// Mitsubishi GX Works2 project: GPF-73G-N2-21110030(220208)   PLC: Q02U

PROGRAM OVEN
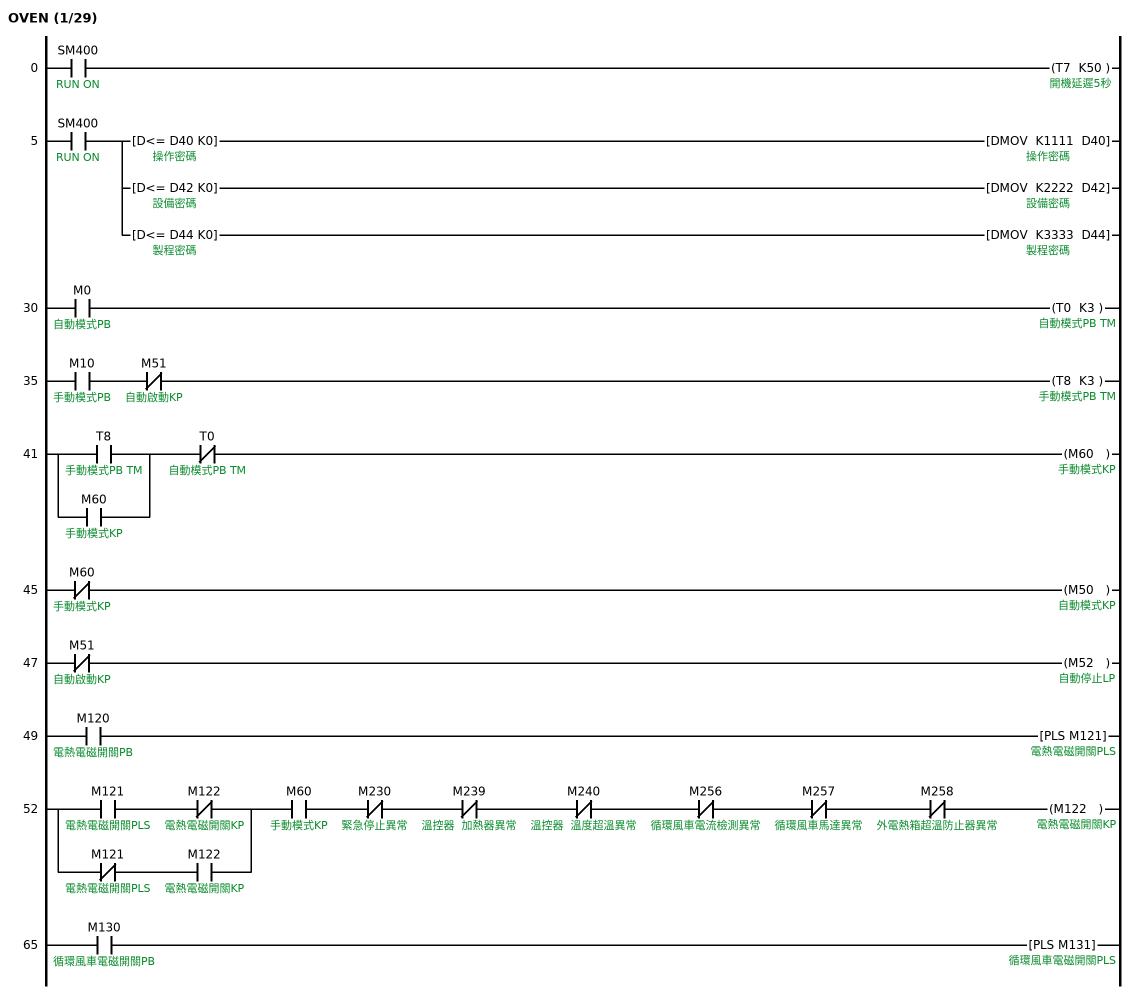
0     LD      SM400  ; RUN ON
      OUT     T7 K50  ; 開機延遲5秒
5     LD      SM400  ; RUN ON
      MPS
      ANDD<=  D40 K0  ; 操作密碼
      DMOV    K1111 D40
      MRD
      ANDD<=  D42 K0  ; 設備密碼
      DMOV    K2222 D42
      MPP
      ANDD<=  D44 K0  ; 製程密碼
      DMOV    K3333 D44
30    LD      M0  ; 自動模式PB
      OUT     T0 K3  ; 自動模式PB TM
35    LD      M10  ; 手動模式PB
      ANI     M51  ; 自動啟動KP
      OUT     T8 K3  ; 手動模式PB TM
41    LD      T8  ; 手動模式PB TM
      OR      M60  ; 手動模式KP
      ANI     T0  ; 自動模式PB TM
      OUT     M60  ; 手動模式KP
45    LDI     M60  ; 手動模式KP
      OUT     M50  ; 自動模式KP
47    LDI     M51  ; 自動啟動KP
      OUT     M52  ; 自動停止LP
49    LD      M120  ; 電熱電磁開關PB
      PLS     M121  ; 電熱電磁開關PLS
52    LD      M121  ; 電熱電磁開關PLS
      ANI     M122  ; 電熱電磁開關KP
      LDI     M121  ; 電熱電磁開關PLS
      AND     M122  ; 電熱電磁開關KP
      ORB
      AND     M60  ; 手動模式KP
      ANI     M230  ; 緊急停止異常
      ANI     M239  ; 溫控器  加熱器異常
      ANI     M240  ; 溫控器  溫度超溫異常
      ANI     M256  ; 循環風車電流檢測異常
      ANI     M257  ; 循環風車馬達異常
      ANI     M258  ; 外電熱箱超溫防止器異常
      OUT     M122  ; 電熱電磁開關KP
65    LD      M130  ; 循環風車電磁開關PB
      PLS     M131  ; 循環風車電磁開關PLS
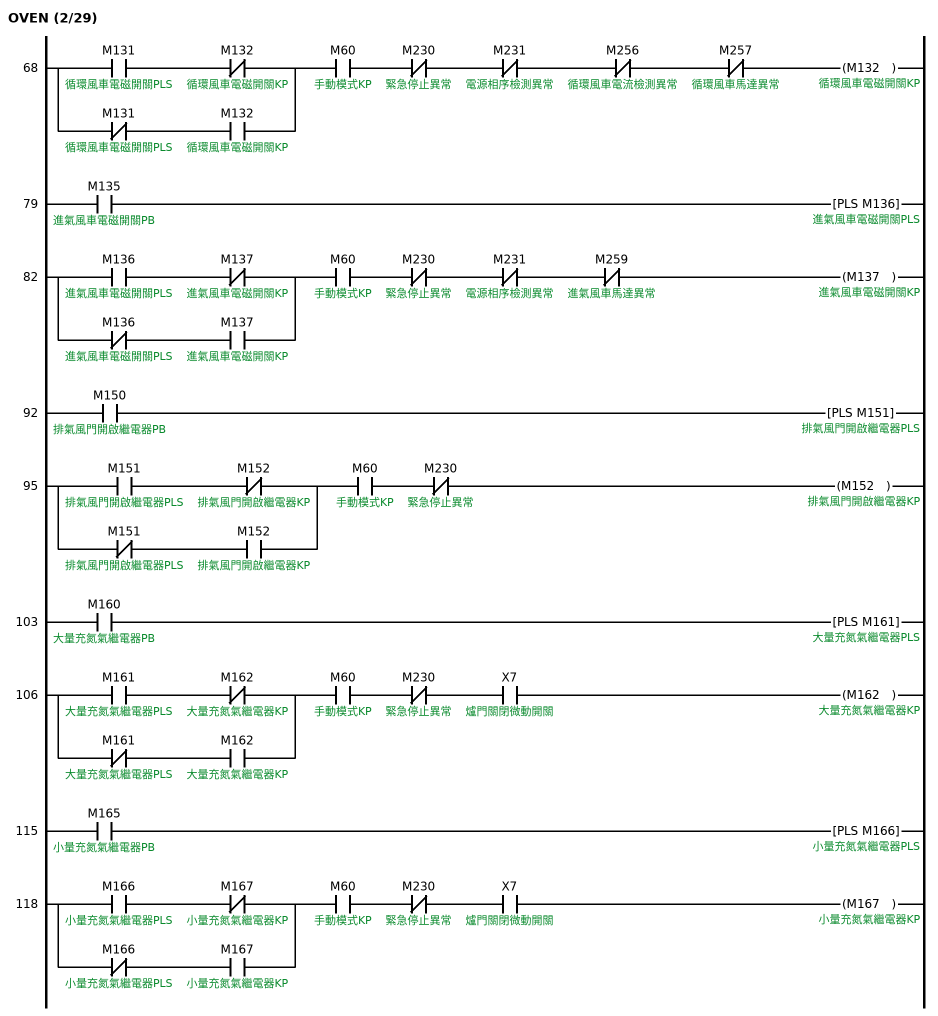
68    LD      M131  ; 循環風車電磁開關PLS
      ANI     M132  ; 循環風車電磁開關KP
      LDI     M131  ; 循環風車電磁開關PLS
      AND     M132  ; 循環風車電磁開關KP
      ORB
      AND     M60  ; 手動模式KP
      ANI     M230  ; 緊急停止異常
      ANI     M231  ; 電源相序檢測異常
      ANI     M256  ; 循環風車電流檢測異常
      ANI     M257  ; 循環風車馬達異常
      OUT     M132  ; 循環風車電磁開關KP
79    LD      M135  ; 進氣風車電磁開關PB
      PLS     M136  ; 進氣風車電磁開關PLS
82    LD      M136  ; 進氣風車電磁開關PLS
      ANI     M137  ; 進氣風車電磁開關KP
      LDI     M136  ; 進氣風車電磁開關PLS
      AND     M137  ; 進氣風車電磁開關KP
      ORB
      AND     M60  ; 手動模式KP
      ANI     M230  ; 緊急停止異常
      ANI     M231  ; 電源相序檢測異常
      ANI     M259  ; 進氣風車馬達異常
      OUT     M137  ; 進氣風車電磁開關KP
92    LD      M150  ; 排氣風門開啟繼電器PB
      PLS     M151  ; 排氣風門開啟繼電器PLS
95    LD      M151  ; 排氣風門開啟繼電器PLS
      ANI     M152  ; 排氣風門開啟繼電器KP
      LDI     M151  ; 排氣風門開啟繼電器PLS
      AND     M152  ; 排氣風門開啟繼電器KP
      ORB
      AND     M60  ; 手動模式KP
      ANI     M230  ; 緊急停止異常
      OUT     M152  ; 排氣風門開啟繼電器KP
103   LD      M160  ; 大量充氮氣繼電器PB
      PLS     M161  ; 大量充氮氣繼電器PLS
106   LD      M161  ; 大量充氮氣繼電器PLS
      ANI     M162  ; 大量充氮氣繼電器KP
      LDI     M161  ; 大量充氮氣繼電器PLS
      AND     M162  ; 大量充氮氣繼電器KP
      ORB
      AND     M60  ; 手動模式KP
      ANI     M230  ; 緊急停止異常
      AND     X7  ; 爐門關閉微動開關
      OUT     M162  ; 大量充氮氣繼電器KP
115   LD      M165  ; 小量充氮氣繼電器PB
      PLS     M166  ; 小量充氮氣繼電器PLS
118   LD      M166  ; 小量充氮氣繼電器PLS
      ANI     M167  ; 小量充氮氣繼電器KP
      LDI     M166  ; 小量充氮氣繼電器PLS
      AND     M167  ; 小量充氮氣繼電器KP
      ORB
      AND     M60  ; 手動模式KP
      ANI     M230  ; 緊急停止異常
      AND     X7  ; 爐門關閉微動開關
      OUT     M167  ; 小量充氮氣繼電器KP
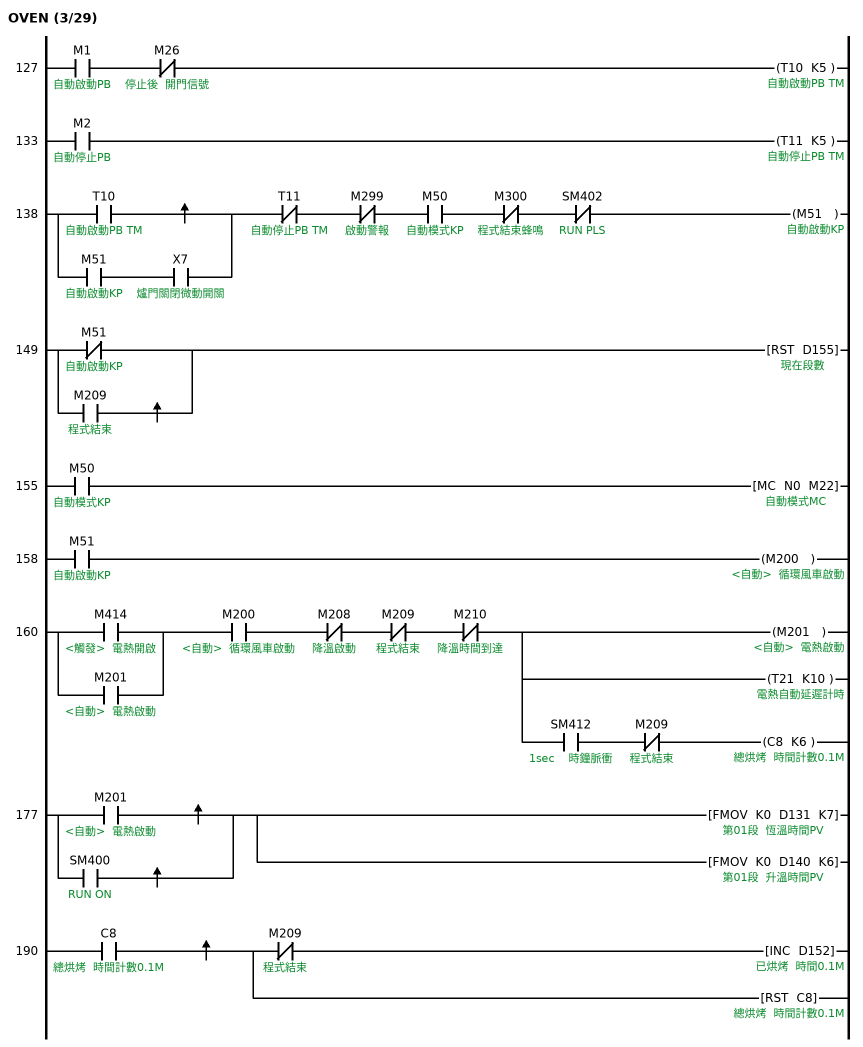
127   LD      M1  ; 自動啟動PB
      ANI     M26  ; 停止後  開門信號
      OUT     T10 K5  ; 自動啟動PB TM
133   LD      M2  ; 自動停止PB
      OUT     T11 K5  ; 自動停止PB TM
138   LD      T10  ; 自動啟動PB TM
      MEP
      LD      M51  ; 自動啟動KP
      AND     X7  ; 爐門關閉微動開關
      ORB
      ANI     T11  ; 自動停止PB TM
      ANI     M299  ; 啟動警報
      AND     M50  ; 自動模式KP
      ANI     M300  ; 程式結束蜂鳴
      ANI     SM402  ; RUN PLS
      OUT     M51  ; 自動啟動KP
149   LDI     M51  ; 自動啟動KP
      LD      M209  ; 程式結束
      MEP
      ORB
      RST     D155  ; 現在段數
155   LD      M50  ; 自動模式KP
      MC      N0 M22  ; 自動模式MC
158   LD      M51  ; 自動啟動KP
      OUT     M200  ; <自動>  循環風車啟動
160   LD      M414  ; <觸發>  電熱開啟
      OR      M201  ; <自動>  電熱啟動
      AND     M200  ; <自動>  循環風車啟動
      ANI     M208  ; 降溫啟動
      ANI     M209  ; 程式結束
      ANI     M210  ; 降溫時間到達
      OUT     M201  ; <自動>  電熱啟動
      OUT     T21 K10  ; 電熱自動延遲計時
      AND     SM412  ; 1sec    時鐘脈衝
      ANI     M209  ; 程式結束
      OUT     C8 K6  ; 總烘烤  時間計數0.1M
177   LD      M201  ; <自動>  電熱啟動
      MEP
      LD      SM400  ; RUN ON
      MEP
      ORB
      FMOV    K0 D131 K7  ; 第01段  恆溫時間PV
      FMOV    K0 D140 K6  ; 第01段  升溫時間PV
190   LD      C8  ; 總烘烤  時間計數0.1M
      MEP
      MPS
      ANI     M209  ; 程式結束
      INC     D152  ; 已烘烤  時間0.1M
      MPP
      RST     C8  ; 總烘烤  時間計數0.1M
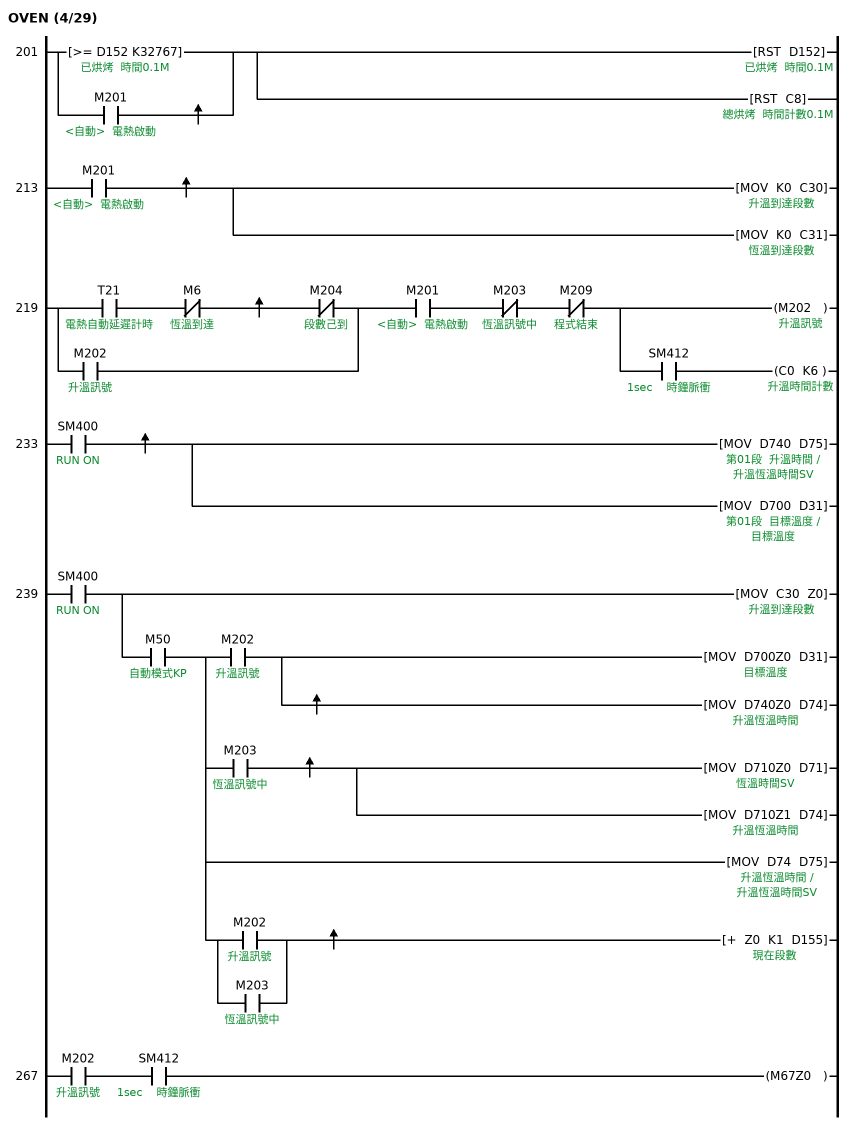
201   LD>=    D152 K32767  ; 已烘烤  時間0.1M
      LD      M201  ; <自動>  電熱啟動
      MEP
      ORB
      RST     D152  ; 已烘烤  時間0.1M
      RST     C8  ; 總烘烤  時間計數0.1M
213   LD      M201  ; <自動>  電熱啟動
      MEP
      MOV     K0 C30  ; 升溫到達段數
      MOV     K0 C31  ; 恆溫到達段數
219   LD      T21  ; 電熱自動延遲計時
      ANI     M6  ; 恆溫到達
      MEP
      ANI     M204  ; 段數己到
      OR      M202  ; 升溫訊號
      AND     M201  ; <自動>  電熱啟動
      ANI     M203  ; 恆溫訊號中
      ANI     M209  ; 程式結束
      OUT     M202  ; 升溫訊號
      AND     SM412  ; 1sec    時鐘脈衝
      OUT     C0 K6  ; 升溫時間計數
233   LD      SM400  ; RUN ON
      MEP
      MOV     D740 D75  ; 第01段  升溫時間 / 升溫恆溫時間SV
      MOV     D700 D31  ; 第01段  目標溫度 / 目標溫度
239   LD      SM400  ; RUN ON
      MOV     C30 Z0
      AND     M50  ; 自動模式KP
      MPS
      AND     M202  ; 升溫訊號
      MOV     D700Z0 D31
      MEP
      MOV     D740Z0 D74  ; 升溫恆溫時間
      MRD
      AND     M203  ; 恆溫訊號中
      MEP
      MOV     D710Z0 D71  ; 恆溫時間SV
      MOV     D710Z1 D74
      MPP
      MOV     D74 D75
      LD      M202  ; 升溫訊號
      OR      M203  ; 恆溫訊號中
      ANB
      MEP
      +       Z0 K1 D155
267   LD      M202  ; 升溫訊號
      AND     SM412  ; 1sec    時鐘脈衝
      OUT     M67Z0
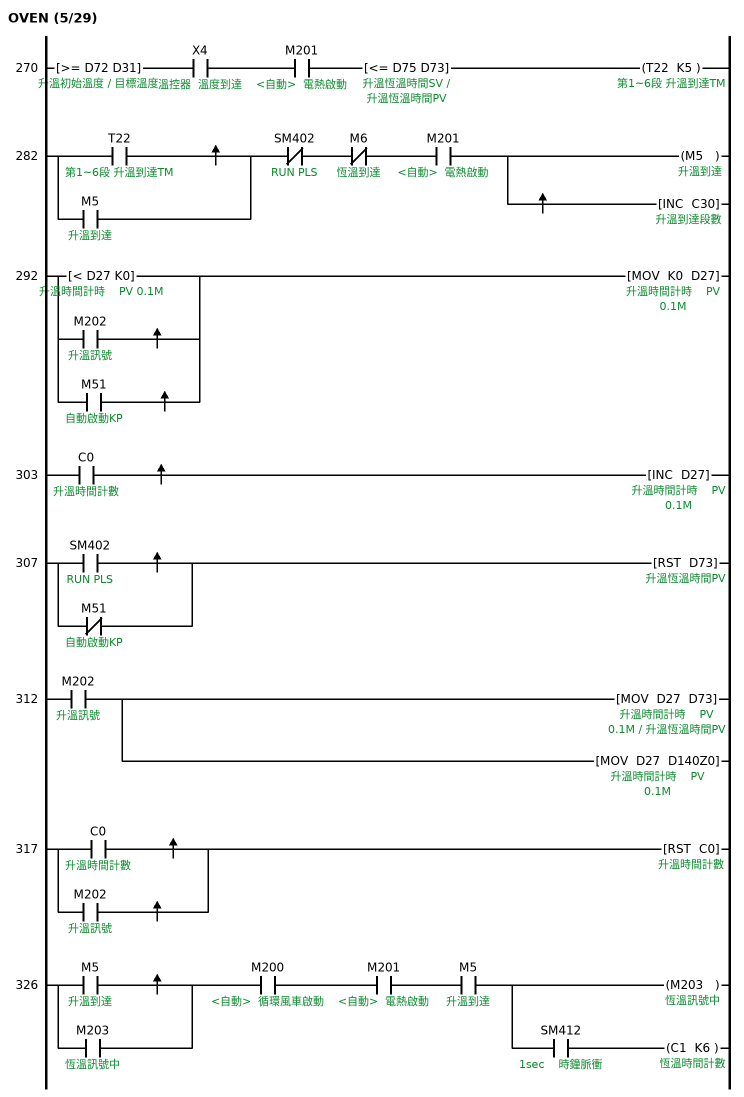
270   LD>=    D72 D31  ; 升溫初始溫度 / 目標溫度
      AND     X4  ; 溫控器  溫度到達
      AND     M201  ; <自動>  電熱啟動
      AND<=   D75 D73  ; 升溫恆溫時間SV / 升溫恆溫時間PV
      OUT     T22 K5  ; 第1~6段 升溫到達TM
282   LD      T22  ; 第1~6段 升溫到達TM
      MEP
      OR      M5  ; 升溫到達
      ANI     SM402  ; RUN PLS
      ANI     M6  ; 恆溫到達
      AND     M201  ; <自動>  電熱啟動
      OUT     M5  ; 升溫到達
      MEP
      INC     C30
292   LD<     D27 K0  ; 升溫時間計時    PV 0.1M
      LD      M202  ; 升溫訊號
      MEP
      ORB
      LD      M51  ; 自動啟動KP
      MEP
      ORB
      MOV     K0 D27
303   LD      C0  ; 升溫時間計數
      MEP
      INC     D27
307   LD      SM402  ; RUN PLS
      MEP
      ORI     M51  ; 自動啟動KP
      RST     D73  ; 升溫恆溫時間PV
312   LD      M202  ; 升溫訊號
      MOV     D27 D73
      MOV     D27 D140Z0
317   LD      C0  ; 升溫時間計數
      MEP
      LD      M202  ; 升溫訊號
      MEP
      ORB
      RST     C0  ; 升溫時間計數
326   LD      M5  ; 升溫到達
      MEP
      OR      M203  ; 恆溫訊號中
      AND     M200  ; <自動>  循環風車啟動
      AND     M201  ; <自動>  電熱啟動
      AND     M5  ; 升溫到達
      OUT     M203  ; 恆溫訊號中
      AND     SM412  ; 1sec    時鐘脈衝
      OUT     C1 K6  ; 恆溫時間計數
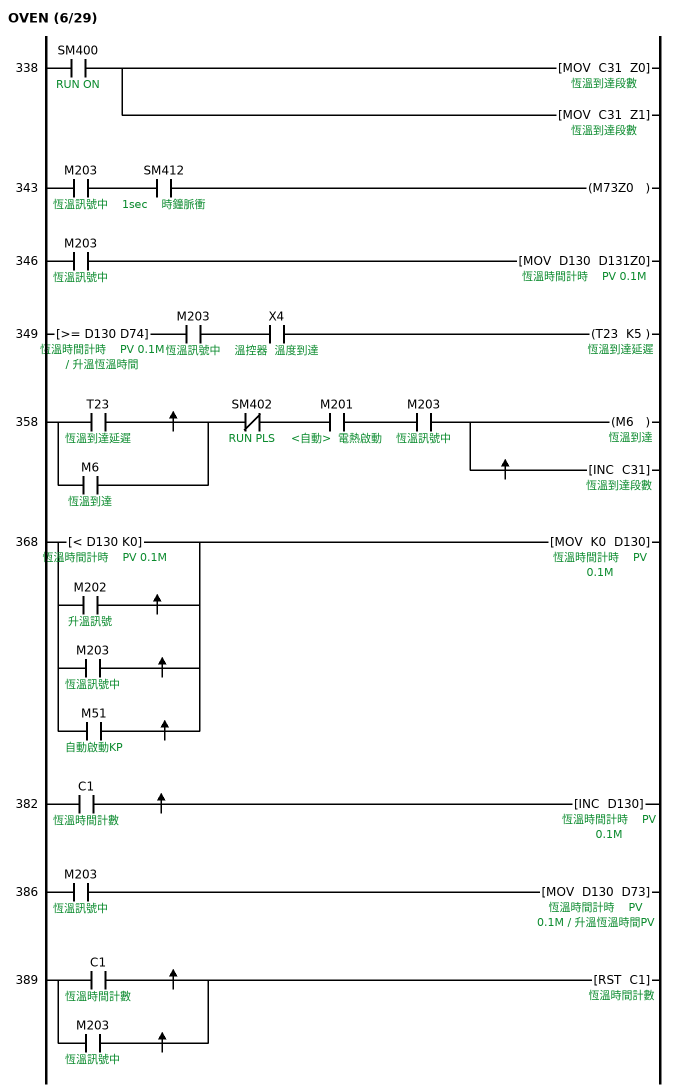
338   LD      SM400  ; RUN ON
      MOV     C31 Z0
      MOV     C31 Z1
343   LD      M203  ; 恆溫訊號中
      AND     SM412  ; 1sec    時鐘脈衝
      OUT     M73Z0
346   LD      M203  ; 恆溫訊號中
      MOV     D130 D131Z0  ; 恆溫時間計時    PV 0.1M
349   LD>=    D130 D74  ; 恆溫時間計時    PV 0.1M / 升溫恆溫時間
      AND     M203  ; 恆溫訊號中
      AND     X4  ; 溫控器  溫度到達
      OUT     T23 K5  ; 恆溫到達延遲
358   LD      T23  ; 恆溫到達延遲
      MEP
      OR      M6  ; 恆溫到達
      ANI     SM402  ; RUN PLS
      AND     M201  ; <自動>  電熱啟動
      AND     M203  ; 恆溫訊號中
      OUT     M6  ; 恆溫到達
      MEP
      INC     C31
368   LD<     D130 K0  ; 恆溫時間計時    PV 0.1M
      LD      M202  ; 升溫訊號
      MEP
      ORB
      LD      M203  ; 恆溫訊號中
      MEP
      ORB
      LD      M51  ; 自動啟動KP
      MEP
      ORB
      MOV     K0 D130
382   LD      C1  ; 恆溫時間計數
      MEP
      INC     D130
386   LD      M203  ; 恆溫訊號中
      MOV     D130 D73
389   LD      C1  ; 恆溫時間計數
      MEP
      LD      M203  ; 恆溫訊號中
      MEP
      ORB
      RST     C1  ; 恆溫時間計數
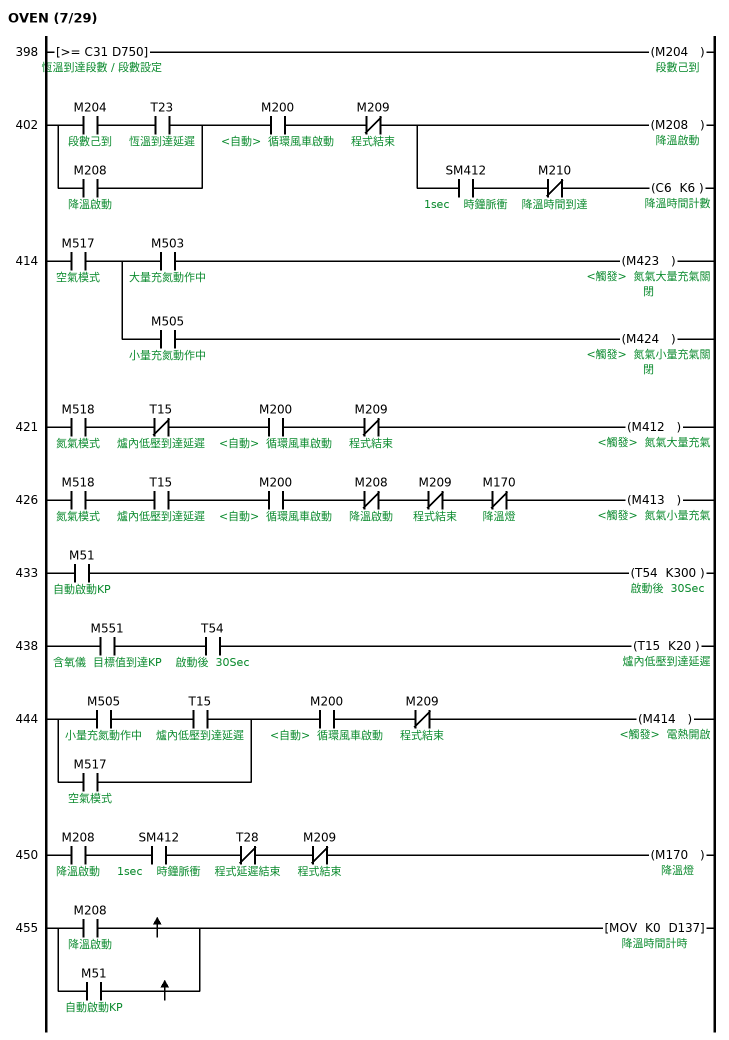
398   LD>=    C31 D750  ; 恆溫到達段數 / 段數設定
      OUT     M204  ; 段數己到
402   LD      M204  ; 段數己到
      AND     T23  ; 恆溫到達延遲
      OR      M208  ; 降溫啟動
      AND     M200  ; <自動>  循環風車啟動
      ANI     M209  ; 程式結束
      OUT     M208  ; 降溫啟動
      AND     SM412  ; 1sec    時鐘脈衝
      ANI     M210  ; 降溫時間到達
      OUT     C6 K6  ; 降溫時間計數
414   LD      M517  ; 空氣模式
      MPS
      AND     M503  ; 大量充氮動作中
      OUT     M423  ; <觸發>  氮氣大量充氣關閉
      MPP
      AND     M505  ; 小量充氮動作中
      OUT     M424  ; <觸發>  氮氣小量充氣關閉
421   LD      M518  ; 氮氣模式
      ANI     T15  ; 爐內低壓到達延遲
      AND     M200  ; <自動>  循環風車啟動
      ANI     M209  ; 程式結束
      OUT     M412  ; <觸發>  氮氣大量充氣
426   LD      M518  ; 氮氣模式
      AND     T15  ; 爐內低壓到達延遲
      AND     M200  ; <自動>  循環風車啟動
      ANI     M208  ; 降溫啟動
      ANI     M209  ; 程式結束
      ANI     M170  ; 降溫燈
      OUT     M413  ; <觸發>  氮氣小量充氣
433   LD      M51  ; 自動啟動KP
      OUT     T54 K300  ; 啟動後  30Sec
438   LD      M551  ; 含氧儀  目標值到達KP
      AND     T54  ; 啟動後  30Sec
      OUT     T15 K20  ; 爐內低壓到達延遲
444   LD      M505  ; 小量充氮動作中
      AND     T15  ; 爐內低壓到達延遲
      OR      M517  ; 空氣模式
      AND     M200  ; <自動>  循環風車啟動
      ANI     M209  ; 程式結束
      OUT     M414  ; <觸發>  電熱開啟
450   LD      M208  ; 降溫啟動
      AND     SM412  ; 1sec    時鐘脈衝
      ANI     T28  ; 程式延遲結束
      ANI     M209  ; 程式結束
      OUT     M170  ; 降溫燈
455   LD      M208  ; 降溫啟動
      MEP
      LD      M51  ; 自動啟動KP
      MEP
      ORB
      MOV     K0 D137  ; 降溫時間計時
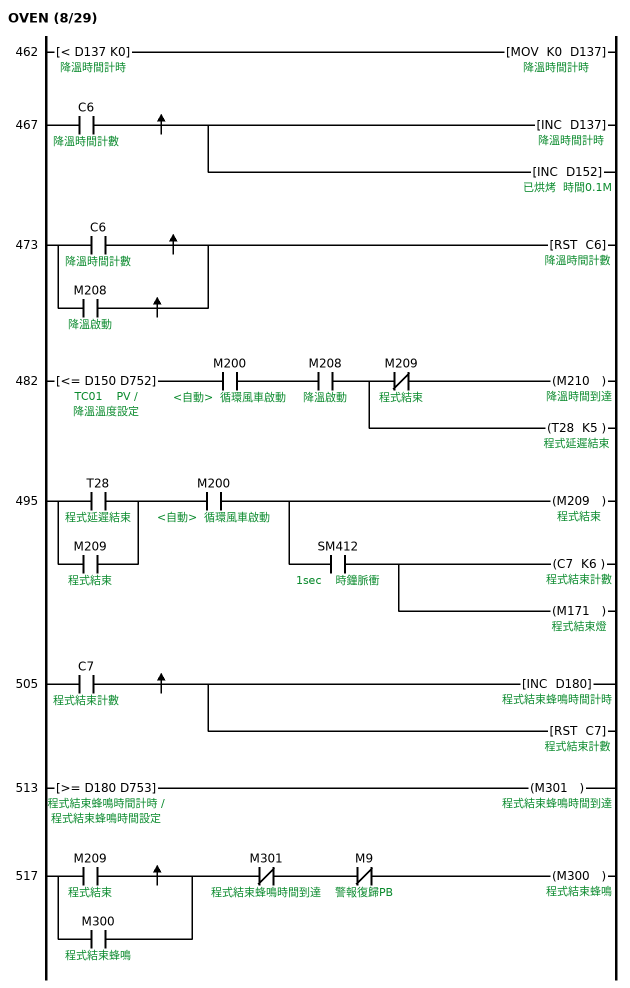
462   LD<     D137 K0  ; 降溫時間計時
      MOV     K0 D137
467   LD      C6  ; 降溫時間計數
      MEP
      INC     D137
      INC     D152
473   LD      C6  ; 降溫時間計數
      MEP
      LD      M208  ; 降溫啟動
      MEP
      ORB
      RST     C6  ; 降溫時間計數
482   LD<=    D150 D752  ; TC01    PV / 降溫溫度設定
      AND     M200  ; <自動>  循環風車啟動
      AND     M208  ; 降溫啟動
      MPS
      ANI     M209  ; 程式結束
      OUT     M210  ; 降溫時間到達
      MPP
      OUT     T28 K5  ; 程式延遲結束
495   LD      T28  ; 程式延遲結束
      OR      M209  ; 程式結束
      AND     M200  ; <自動>  循環風車啟動
      OUT     M209  ; 程式結束
      AND     SM412  ; 1sec    時鐘脈衝
      OUT     C7 K6  ; 程式結束計數
      OUT     M171  ; 程式結束燈
505   LD      C7  ; 程式結束計數
      MEP
      INC     D180  ; 程式結束蜂鳴時間計時
      RST     C7  ; 程式結束計數
513   LD>=    D180 D753  ; 程式結束蜂鳴時間計時 / 程式結束蜂鳴時間設定
      OUT     M301  ; 程式結束蜂鳴時間到達
517   LD      M209  ; 程式結束
      MEP
      OR      M300  ; 程式結束蜂鳴
      ANI     M301  ; 程式結束蜂鳴時間到達
      ANI     M9  ; 警報復歸PB
      OUT     M300  ; 程式結束蜂鳴
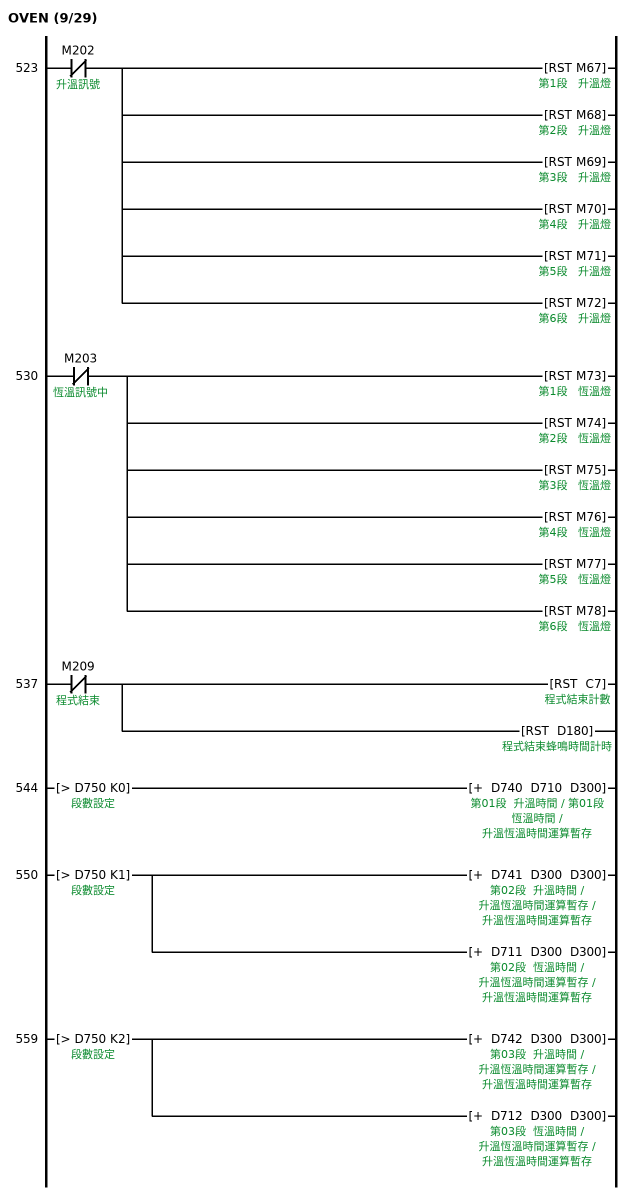
523   LDI     M202  ; 升溫訊號
      RST     M67  ; 第1段   升溫燈
      RST     M68  ; 第2段   升溫燈
      RST     M69  ; 第3段   升溫燈
      RST     M70  ; 第4段   升溫燈
      RST     M71  ; 第5段   升溫燈
      RST     M72  ; 第6段   升溫燈
530   LDI     M203  ; 恆溫訊號中
      RST     M73  ; 第1段   恆溫燈
      RST     M74  ; 第2段   恆溫燈
      RST     M75  ; 第3段   恆溫燈
      RST     M76  ; 第4段   恆溫燈
      RST     M77  ; 第5段   恆溫燈
      RST     M78  ; 第6段   恆溫燈
537   LDI     M209  ; 程式結束
      RST     C7  ; 程式結束計數
      RST     D180  ; 程式結束蜂鳴時間計時
544   LD>     D750 K0  ; 段數設定
      +       D740 D710 D300  ; 第01段  恆溫時間 / 升溫恆溫時間運算暫存
550   LD>     D750 K1  ; 段數設定
      +       D741 D300 D300  ; 第02段  升溫時間
      +       D711 D300 D300  ; 第02段  恆溫時間
559   LD>     D750 K2  ; 段數設定
      +       D742 D300 D300  ; 第03段  升溫時間
      +       D712 D300 D300  ; 第03段  恆溫時間
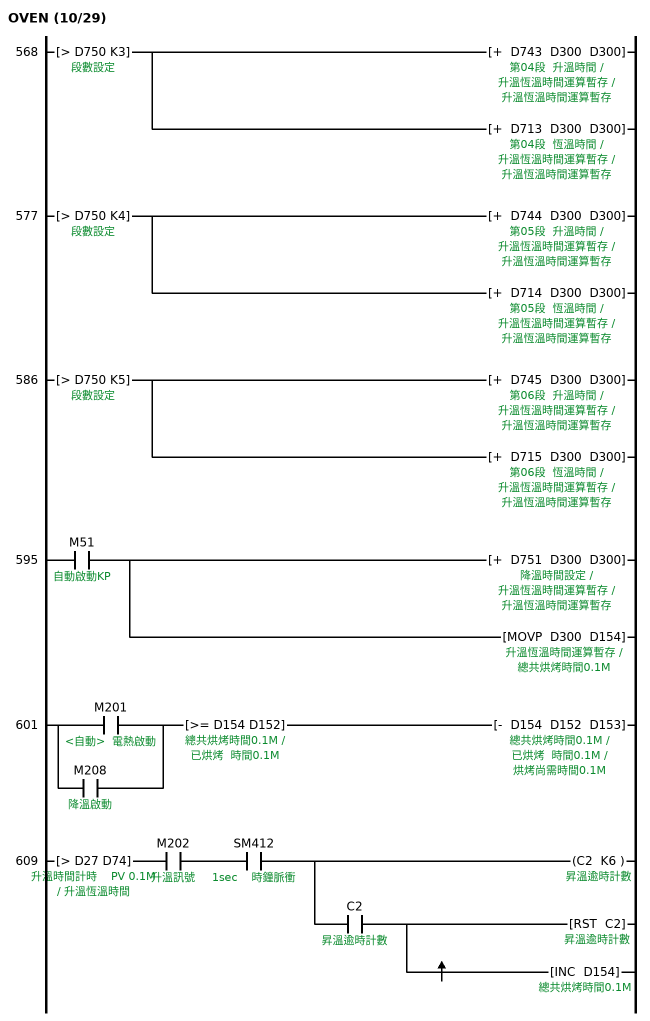
568   LD>     D750 K3  ; 段數設定
      +       D743 D300 D300  ; 第04段  升溫時間
      +       D713 D300 D300  ; 第04段  恆溫時間
577   LD>     D750 K4  ; 段數設定
      +       D744 D300 D300  ; 第05段  升溫時間
      +       D714 D300 D300  ; 第05段  恆溫時間
586   LD>     D750 K5  ; 段數設定
      +       D745 D300 D300  ; 第06段  升溫時間
      +       D715 D300 D300  ; 第06段  恆溫時間
595   LD      M51  ; 自動啟動KP
      +       D751 D300 D300  ; 降溫時間設定
      MOVP    D300 D154  ; 總共烘烤時間0.1M
601   LD      M201  ; <自動>  電熱啟動
      OR      M208  ; 降溫啟動
      AND>=   D154 D152  ; 總共烘烤時間0.1M / 已烘烤  時間0.1M
      -       D154 D152 D153  ; 烘烤尚需時間0.1M
609   LD>     D27 D74  ; 升溫時間計時    PV 0.1M / 升溫恆溫時間
      AND     M202  ; 升溫訊號
      AND     SM412  ; 1sec    時鐘脈衝
      OUT     C2 K6  ; 昇溫逾時計數
      AND     C2  ; 昇溫逾時計數
      RST     C2  ; 昇溫逾時計數
      MEP
      INC     D154
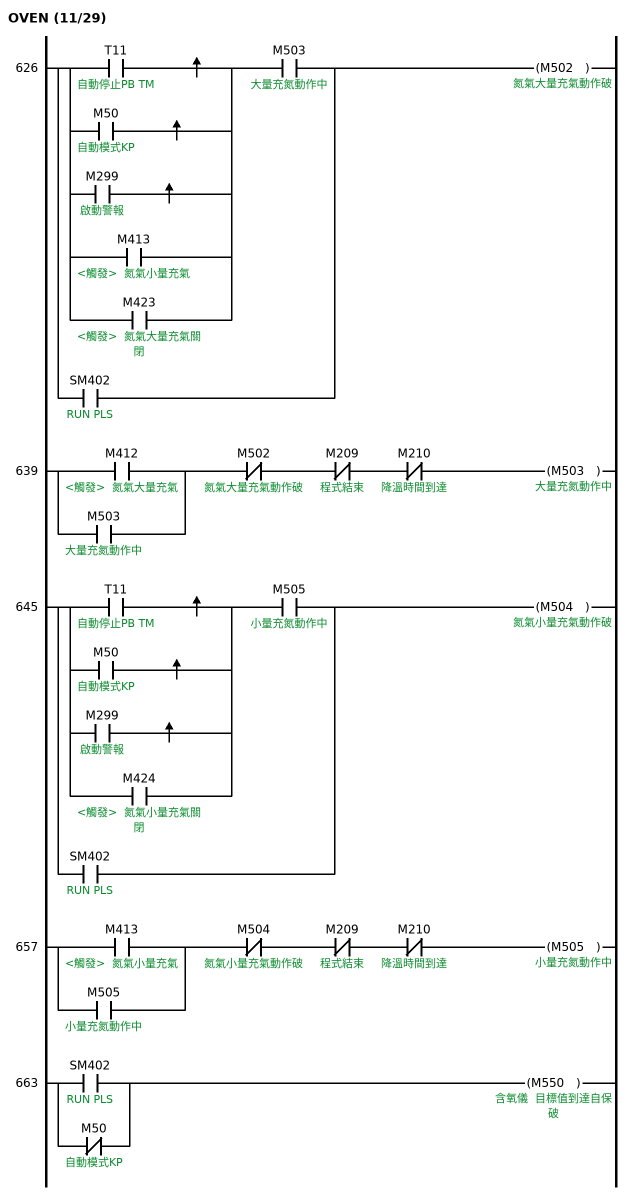
626   LD      T11  ; 自動停止PB TM
      MEP
      LD      M50  ; 自動模式KP
      MEP
      ORB
      LD      M299  ; 啟動警報
      MEP
      ORB
      OR      M413  ; <觸發>  氮氣小量充氣
      OR      M423  ; <觸發>  氮氣大量充氣關閉
      AND     M503  ; 大量充氮動作中
      OR      SM402  ; RUN PLS
      OUT     M502  ; 氮氣大量充氣動作破
639   LD      M412  ; <觸發>  氮氣大量充氣
      OR      M503  ; 大量充氮動作中
      ANI     M502  ; 氮氣大量充氣動作破
      ANI     M209  ; 程式結束
      ANI     M210  ; 降溫時間到達
      OUT     M503  ; 大量充氮動作中
645   LD      T11  ; 自動停止PB TM
      MEP
      LD      M50  ; 自動模式KP
      MEP
      ORB
      LD      M299  ; 啟動警報
      MEP
      ORB
      OR      M424  ; <觸發>  氮氣小量充氣關閉
      AND     M505  ; 小量充氮動作中
      OR      SM402  ; RUN PLS
      OUT     M504  ; 氮氣小量充氣動作破
657   LD      M413  ; <觸發>  氮氣小量充氣
      OR      M505  ; 小量充氮動作中
      ANI     M504  ; 氮氣小量充氣動作破
      ANI     M209  ; 程式結束
      ANI     M210  ; 降溫時間到達
      OUT     M505  ; 小量充氮動作中
663   LD      SM402  ; RUN PLS
      ORI     M50  ; 自動模式KP
      OUT     M550  ; 含氧儀  目標值到達自保破
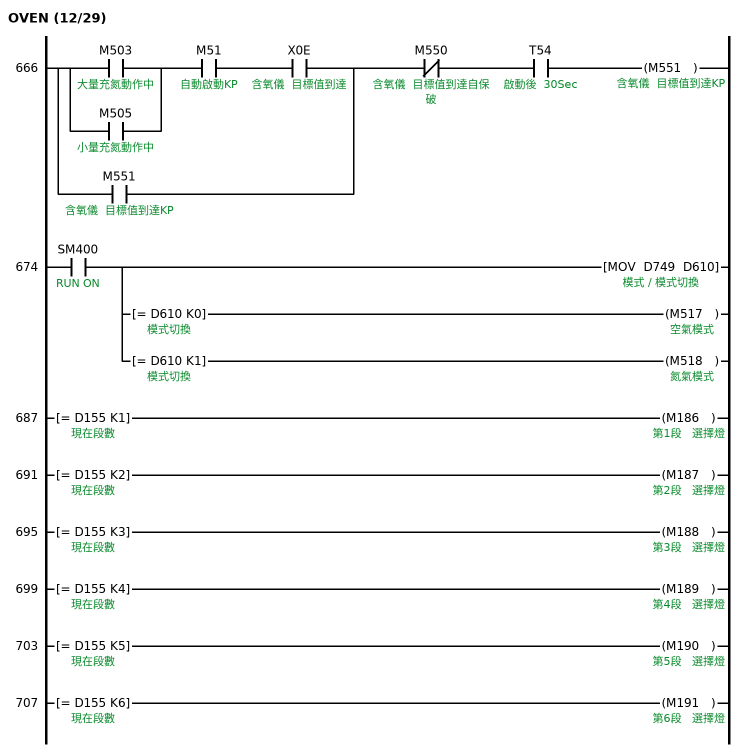
666   LD      M503  ; 大量充氮動作中
      OR      M505  ; 小量充氮動作中
      AND     M51  ; 自動啟動KP
      AND     X0E  ; 含氧儀  目標值到達
      OR      M551  ; 含氧儀  目標值到達KP
      ANI     M550  ; 含氧儀  目標值到達自保破
      AND     T54  ; 啟動後  30Sec
      OUT     M551  ; 含氧儀  目標值到達KP
674   LD      SM400  ; RUN ON
      MOV     D749 D610  ; 模式 / 模式切換
      MPS
      AND=    D610 K0  ; 模式切換
      OUT     M517  ; 空氣模式
      MPP
      AND=    D610 K1  ; 模式切換
      OUT     M518  ; 氮氣模式
687   LD=     D155 K1  ; 現在段數
      OUT     M186  ; 第1段   選擇燈
691   LD=     D155 K2  ; 現在段數
      OUT     M187  ; 第2段   選擇燈
695   LD=     D155 K3  ; 現在段數
      OUT     M188  ; 第3段   選擇燈
699   LD=     D155 K4  ; 現在段數
      OUT     M189  ; 第4段   選擇燈
703   LD=     D155 K5  ; 現在段數
      OUT     M190  ; 第5段   選擇燈
707   LD=     D155 K6  ; 現在段數
      OUT     M191  ; 第6段   選擇燈
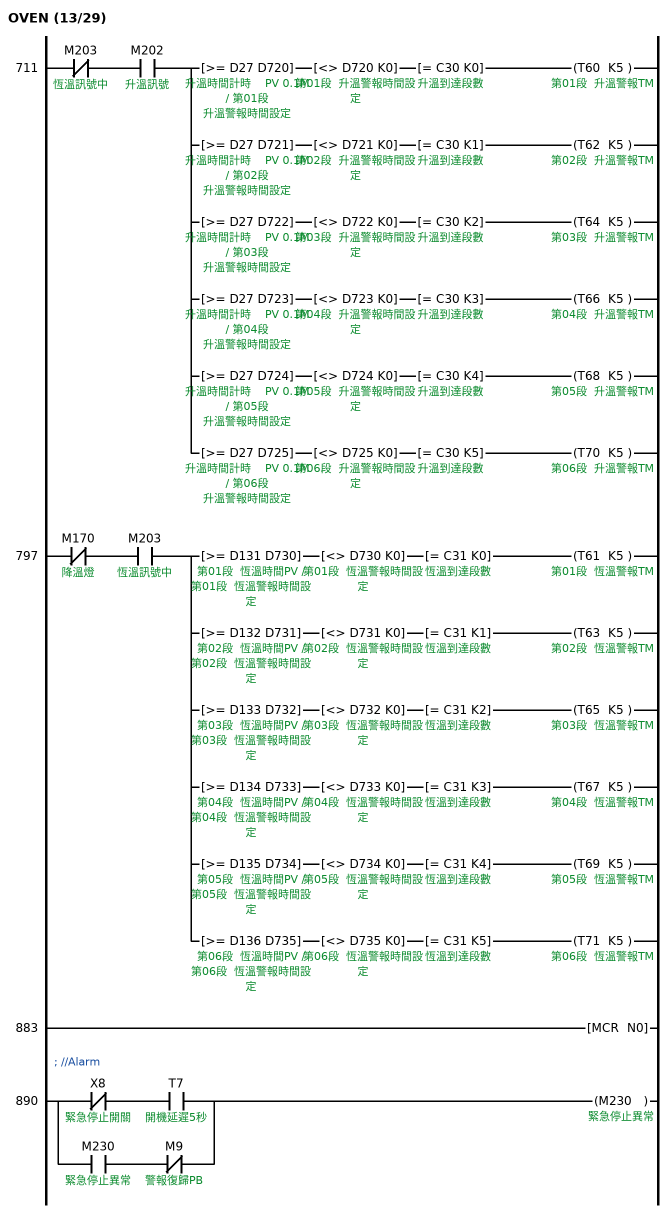
711   LDI     M203  ; 恆溫訊號中
      AND     M202  ; 升溫訊號
      MPS
      AND>=   D27 D720  ; 升溫時間計時    PV 0.1M / 第01段  升溫警報時間設定
      AND<>   D720 K0  ; 第01段  升溫警報時間設定
      AND=    C30 K0  ; 升溫到達段數
      OUT     T60 K5  ; 第01段  升溫警報TM
      MRD
      AND>=   D27 D721  ; 升溫時間計時    PV 0.1M / 第02段  升溫警報時間設定
      AND<>   D721 K0  ; 第02段  升溫警報時間設定
      AND=    C30 K1  ; 升溫到達段數
      OUT     T62 K5  ; 第02段  升溫警報TM
      MRD
      AND>=   D27 D722  ; 升溫時間計時    PV 0.1M / 第03段  升溫警報時間設定
      AND<>   D722 K0  ; 第03段  升溫警報時間設定
      AND=    C30 K2  ; 升溫到達段數
      OUT     T64 K5  ; 第03段  升溫警報TM
      MRD
      AND>=   D27 D723  ; 升溫時間計時    PV 0.1M / 第04段  升溫警報時間設定
      AND<>   D723 K0  ; 第04段  升溫警報時間設定
      AND=    C30 K3  ; 升溫到達段數
      OUT     T66 K5  ; 第04段  升溫警報TM
      MRD
      AND>=   D27 D724  ; 升溫時間計時    PV 0.1M / 第05段  升溫警報時間設定
      AND<>   D724 K0  ; 第05段  升溫警報時間設定
      AND=    C30 K4  ; 升溫到達段數
      OUT     T68 K5  ; 第05段  升溫警報TM
      MPP
      AND>=   D27 D725  ; 升溫時間計時    PV 0.1M / 第06段  升溫警報時間設定
      AND<>   D725 K0  ; 第06段  升溫警報時間設定
      AND=    C30 K5  ; 升溫到達段數
      OUT     T70 K5  ; 第06段  升溫警報TM
797   LDI     M170  ; 降溫燈
      AND     M203  ; 恆溫訊號中
      MPS
      AND>=   D131 D730  ; 第01段  恆溫時間PV / 第01段  恆溫警報時間設定
      AND<>   D730 K0  ; 第01段  恆溫警報時間設定
      AND=    C31 K0  ; 恆溫到達段數
      OUT     T61 K5  ; 第01段  恆溫警報TM
      MRD
      AND>=   D132 D731  ; 第02段  恆溫時間PV / 第02段  恆溫警報時間設定
      AND<>   D731 K0  ; 第02段  恆溫警報時間設定
      AND=    C31 K1  ; 恆溫到達段數
      OUT     T63 K5  ; 第02段  恆溫警報TM
      MRD
      AND>=   D133 D732  ; 第03段  恆溫時間PV / 第03段  恆溫警報時間設定
      AND<>   D732 K0  ; 第03段  恆溫警報時間設定
      AND=    C31 K2  ; 恆溫到達段數
      OUT     T65 K5  ; 第03段  恆溫警報TM
      MRD
      AND>=   D134 D733  ; 第04段  恆溫時間PV / 第04段  恆溫警報時間設定
      AND<>   D733 K0  ; 第04段  恆溫警報時間設定
      AND=    C31 K3  ; 恆溫到達段數
      OUT     T67 K5  ; 第04段  恆溫警報TM
      MRD
      AND>=   D135 D734  ; 第05段  恆溫時間PV / 第05段  恆溫警報時間設定
      AND<>   D734 K0  ; 第05段  恆溫警報時間設定
      AND=    C31 K4  ; 恆溫到達段數
      OUT     T69 K5  ; 第05段  恆溫警報TM
      MPP
      AND>=   D136 D735  ; 第06段  恆溫時間PV / 第06段  恆溫警報時間設定
      AND<>   D735 K0  ; 第06段  恆溫警報時間設定
      AND=    C31 K5  ; 恆溫到達段數
      OUT     T71 K5  ; 第06段  恆溫警報TM
883   MCR     N0
; //Alarm
890   LDI     X8  ; 緊急停止開關
      AND     T7  ; 開機延遲5秒
      LD      M230  ; 緊急停止異常
      ANI     M9  ; 警報復歸PB
      ORB
      OUT     M230  ; 緊急停止異常
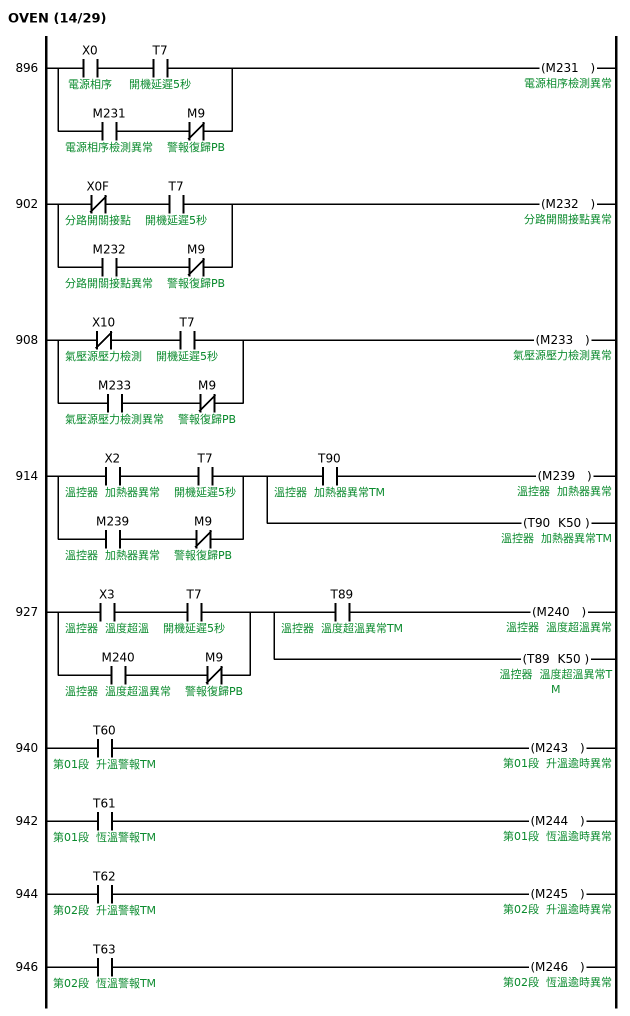
896   LD      X0  ; 電源相序
      AND     T7  ; 開機延遲5秒
      LD      M231  ; 電源相序檢測異常
      ANI     M9  ; 警報復歸PB
      ORB
      OUT     M231  ; 電源相序檢測異常
902   LDI     X0F  ; 分路開關接點
      AND     T7  ; 開機延遲5秒
      LD      M232  ; 分路開關接點異常
      ANI     M9  ; 警報復歸PB
      ORB
      OUT     M232  ; 分路開關接點異常
908   LDI     X10  ; 氣壓源壓力檢測
      AND     T7  ; 開機延遲5秒
      LD      M233  ; 氣壓源壓力檢測異常
      ANI     M9  ; 警報復歸PB
      ORB
      OUT     M233  ; 氣壓源壓力檢測異常
914   LD      X2  ; 溫控器  加熱器異常
      AND     T7  ; 開機延遲5秒
      LD      M239  ; 溫控器  加熱器異常
      ANI     M9  ; 警報復歸PB
      ORB
      MPS
      AND     T90  ; 溫控器  加熱器異常TM
      OUT     M239  ; 溫控器  加熱器異常
      MPP
      OUT     T90 K50  ; 溫控器  加熱器異常TM
927   LD      X3  ; 溫控器  溫度超溫
      AND     T7  ; 開機延遲5秒
      LD      M240  ; 溫控器  溫度超溫異常
      ANI     M9  ; 警報復歸PB
      ORB
      MPS
      AND     T89  ; 溫控器  溫度超溫異常TM
      OUT     M240  ; 溫控器  溫度超溫異常
      MPP
      OUT     T89 K50  ; 溫控器  溫度超溫異常TM
940   LD      T60  ; 第01段  升溫警報TM
      OUT     M243  ; 第01段  升溫逾時異常
942   LD      T61  ; 第01段  恆溫警報TM
      OUT     M244  ; 第01段  恆溫逾時異常
944   LD      T62  ; 第02段  升溫警報TM
      OUT     M245  ; 第02段  升溫逾時異常
946   LD      T63  ; 第02段  恆溫警報TM
      OUT     M246  ; 第02段  恆溫逾時異常
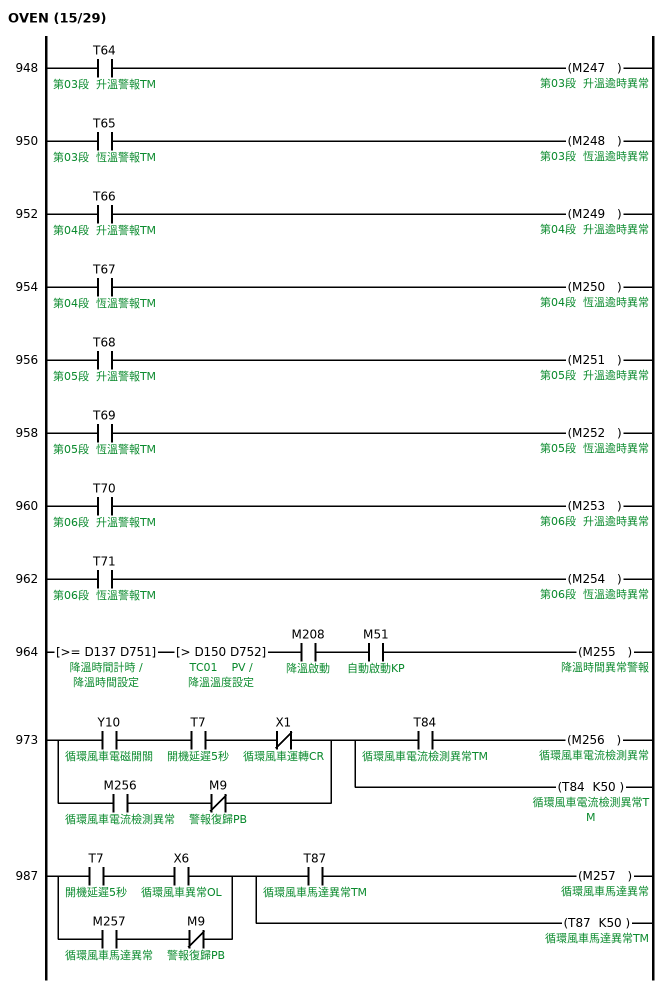
948   LD      T64  ; 第03段  升溫警報TM
      OUT     M247  ; 第03段  升溫逾時異常
950   LD      T65  ; 第03段  恆溫警報TM
      OUT     M248  ; 第03段  恆溫逾時異常
952   LD      T66  ; 第04段  升溫警報TM
      OUT     M249  ; 第04段  升溫逾時異常
954   LD      T67  ; 第04段  恆溫警報TM
      OUT     M250  ; 第04段  恆溫逾時異常
956   LD      T68  ; 第05段  升溫警報TM
      OUT     M251  ; 第05段  升溫逾時異常
958   LD      T69  ; 第05段  恆溫警報TM
      OUT     M252  ; 第05段  恆溫逾時異常
960   LD      T70  ; 第06段  升溫警報TM
      OUT     M253  ; 第06段  升溫逾時異常
962   LD      T71  ; 第06段  恆溫警報TM
      OUT     M254  ; 第06段  恆溫逾時異常
964   LD>=    D137 D751  ; 降溫時間計時 / 降溫時間設定
      AND>    D150 D752  ; TC01    PV / 降溫溫度設定
      AND     M208  ; 降溫啟動
      AND     M51  ; 自動啟動KP
      OUT     M255  ; 降溫時間異常警報
973   LD      Y10  ; 循環風車電磁開關
      AND     T7  ; 開機延遲5秒
      ANI     X1  ; 循環風車運轉CR
      LD      M256  ; 循環風車電流檢測異常
      ANI     M9  ; 警報復歸PB
      ORB
      MPS
      AND     T84  ; 循環風車電流檢測異常TM
      OUT     M256  ; 循環風車電流檢測異常
      MPP
      OUT     T84 K50  ; 循環風車電流檢測異常TM
987   LD      T7  ; 開機延遲5秒
      AND     X6  ; 循環風車異常OL
      LD      M257  ; 循環風車馬達異常
      ANI     M9  ; 警報復歸PB
      ORB
      MPS
      AND     T87  ; 循環風車馬達異常TM
      OUT     M257  ; 循環風車馬達異常
      MPP
      OUT     T87 K50  ; 循環風車馬達異常TM
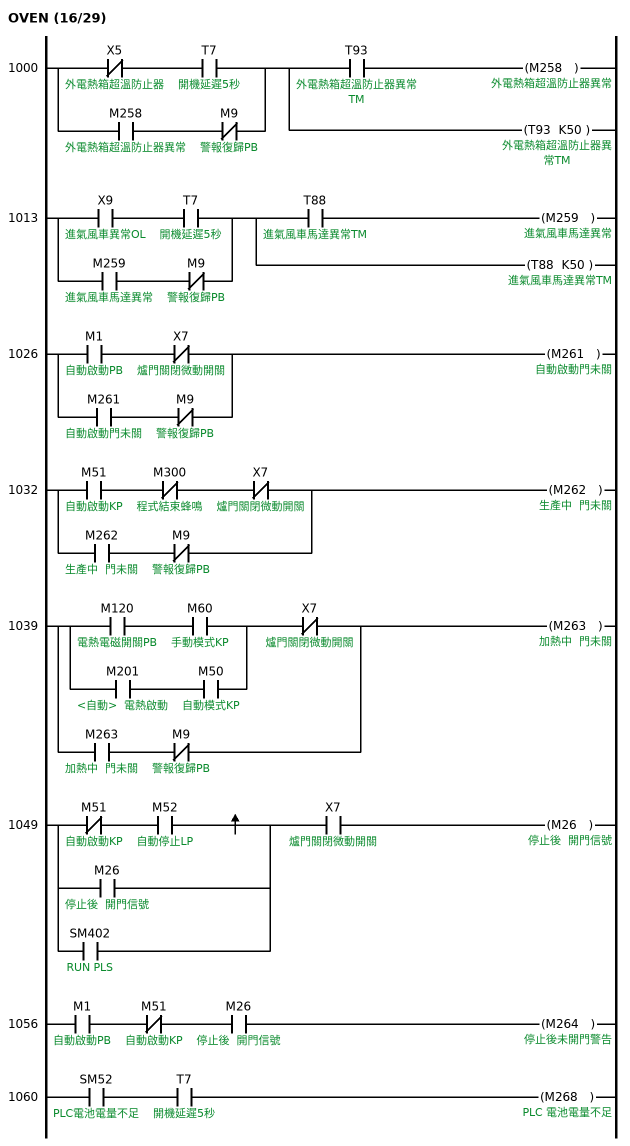
1000  LDI     X5  ; 外電熱箱超溫防止器
      AND     T7  ; 開機延遲5秒
      LD      M258  ; 外電熱箱超溫防止器異常
      ANI     M9  ; 警報復歸PB
      ORB
      MPS
      AND     T93  ; 外電熱箱超溫防止器異常TM
      OUT     M258  ; 外電熱箱超溫防止器異常
      MPP
      OUT     T93 K50  ; 外電熱箱超溫防止器異常TM
1013  LD      X9  ; 進氣風車異常OL
      AND     T7  ; 開機延遲5秒
      LD      M259  ; 進氣風車馬達異常
      ANI     M9  ; 警報復歸PB
      ORB
      MPS
      AND     T88  ; 進氣風車馬達異常TM
      OUT     M259  ; 進氣風車馬達異常
      MPP
      OUT     T88 K50  ; 進氣風車馬達異常TM
1026  LD      M1  ; 自動啟動PB
      ANI     X7  ; 爐門關閉微動開關
      LD      M261  ; 自動啟動門未關
      ANI     M9  ; 警報復歸PB
      ORB
      OUT     M261  ; 自動啟動門未關
1032  LD      M51  ; 自動啟動KP
      ANI     M300  ; 程式結束蜂鳴
      ANI     X7  ; 爐門關閉微動開關
      LD      M262  ; 生產中  門未關
      ANI     M9  ; 警報復歸PB
      ORB
      OUT     M262  ; 生產中  門未關
1039  LD      M120  ; 電熱電磁開關PB
      AND     M60  ; 手動模式KP
      LD      M201  ; <自動>  電熱啟動
      AND     M50  ; 自動模式KP
      ORB
      ANI     X7  ; 爐門關閉微動開關
      LD      M263  ; 加熱中  門未關
      ANI     M9  ; 警報復歸PB
      ORB
      OUT     M263  ; 加熱中  門未關
1049  LDI     M51  ; 自動啟動KP
      AND     M52  ; 自動停止LP
      MEP
      OR      M26  ; 停止後  開門信號
      OR      SM402  ; RUN PLS
      AND     X7  ; 爐門關閉微動開關
      OUT     M26  ; 停止後  開門信號
1056  LD      M1  ; 自動啟動PB
      ANI     M51  ; 自動啟動KP
      AND     M26  ; 停止後  開門信號
      OUT     M264  ; 停止後未開門警告
1060  LD      SM52  ; PLC電池電量不足
      AND     T7  ; 開機延遲5秒
      OUT     M268  ; PLC 電池電量不足
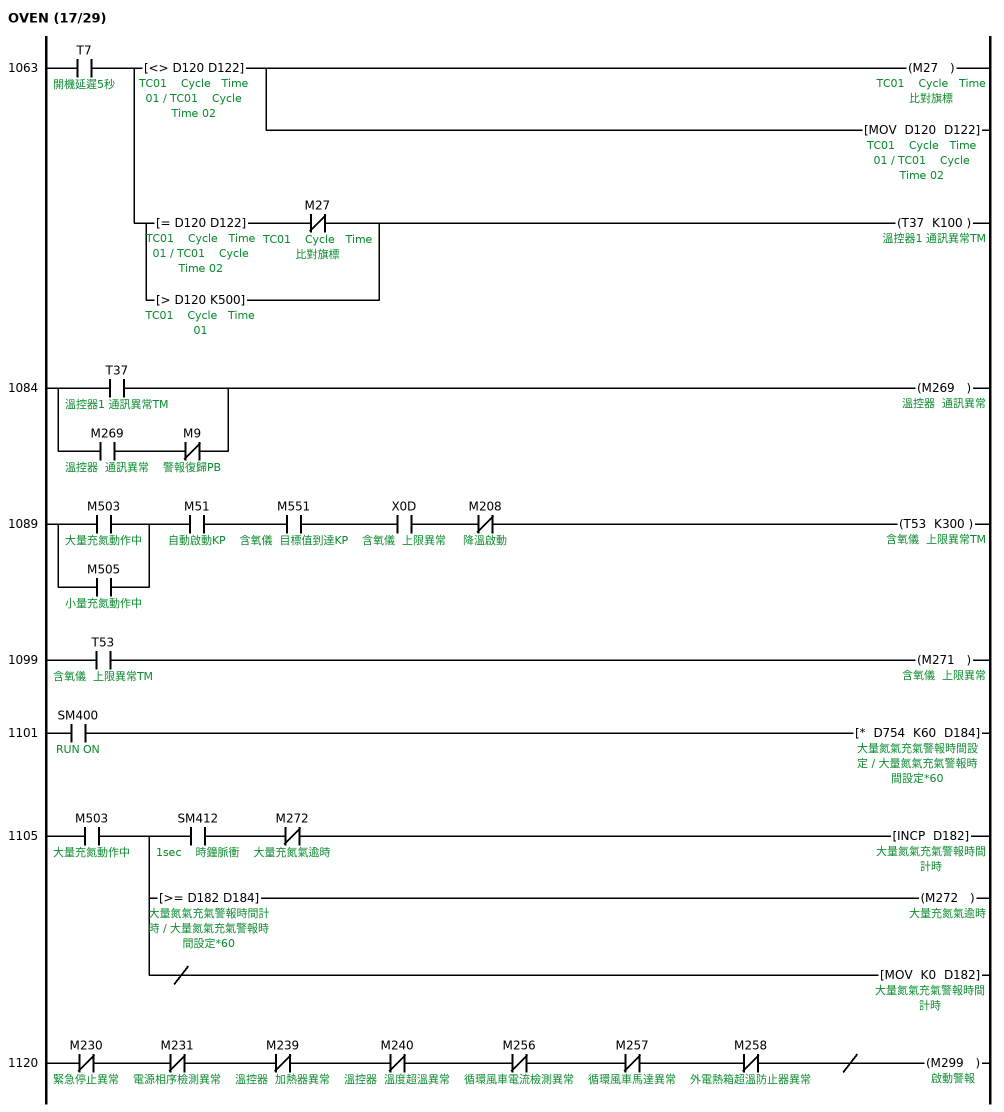
1063  LD      T7  ; 開機延遲5秒
      MPS
      AND<>   D120 D122  ; TC01    Cycle   Time 01 / TC01    Cycle   Time 02
      OUT     M27  ; TC01    Cycle   Time    比對旗標
      MOV     D120 D122
      MPP
      LD=     D120 D122  ; TC01    Cycle   Time 01 / TC01    Cycle   Time 02
      ANI     M27  ; TC01    Cycle   Time    比對旗標
      OR>     D120 K500  ; TC01    Cycle   Time 01
      ANB
      OUT     T37 K100  ; 溫控器1 通訊異常TM
1084  LD      T37  ; 溫控器1 通訊異常TM
      LD      M269  ; 溫控器  通訊異常
      ANI     M9  ; 警報復歸PB
      ORB
      OUT     M269  ; 溫控器  通訊異常
1089  LD      M503  ; 大量充氮動作中
      OR      M505  ; 小量充氮動作中
      AND     M51  ; 自動啟動KP
      AND     M551  ; 含氧儀  目標值到達KP
      AND     X0D  ; 含氧儀  上限異常
      ANI     M208  ; 降溫啟動
      OUT     T53 K300  ; 含氧儀  上限異常TM
1099  LD      T53  ; 含氧儀  上限異常TM
      OUT     M271  ; 含氧儀  上限異常
1101  LD      SM400  ; RUN ON
      *       D754 K60 D184  ; 大量氮氣充氣警報時間設定 / 大量氮氣充氣警報時間設定*60
1105  LD      M503  ; 大量充氮動作中
      MPS
      AND     SM412  ; 1sec    時鐘脈衝
      ANI     M272  ; 大量充氮氣逾時
      INCP    D182  ; 大量氮氣充氣警報時間計時
      MRD
      AND>=   D182 D184  ; 大量氮氣充氣警報時間計時 / 大量氮氣充氣警報時間設定*60
      OUT     M272  ; 大量充氮氣逾時
      MPP
      INV
      MOV     K0 D182
1120  LDI     M230  ; 緊急停止異常
      ANI     M231  ; 電源相序檢測異常
      ANI     M239  ; 溫控器  加熱器異常
      ANI     M240  ; 溫控器  溫度超溫異常
      ANI     M256  ; 循環風車電流檢測異常
      ANI     M257  ; 循環風車馬達異常
      ANI     M258  ; 外電熱箱超溫防止器異常
      INV
      OUT     M299  ; 啟動警報
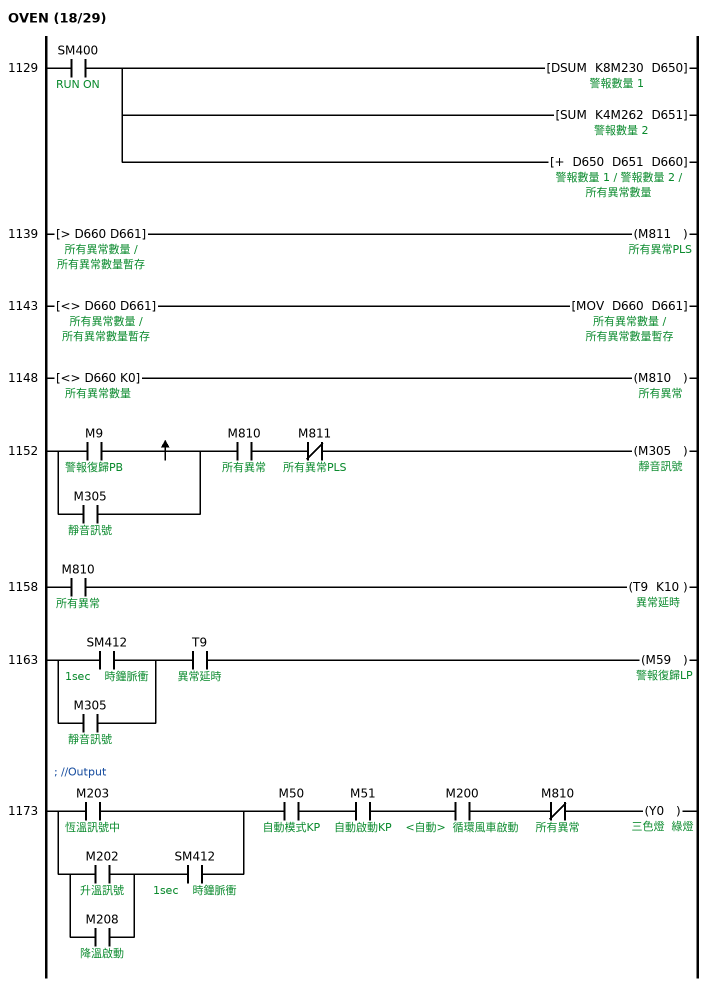
1129  LD      SM400  ; RUN ON
      DSUM    K8M230 D650  ; 警報數量 1
      SUM     K4M262 D651  ; 警報數量 2
      +       D650 D651 D660  ; 所有異常數量
1139  LD>     D660 D661  ; 所有異常數量 / 所有異常數量暫存
      OUT     M811  ; 所有異常PLS
1143  LD<>    D660 D661  ; 所有異常數量 / 所有異常數量暫存
      MOV     D660 D661
1148  LD<>    D660 K0  ; 所有異常數量
      OUT     M810  ; 所有異常
1152  LD      M9  ; 警報復歸PB
      MEP
      OR      M305  ; 靜音訊號
      AND     M810  ; 所有異常
      ANI     M811  ; 所有異常PLS
      OUT     M305  ; 靜音訊號
1158  LD      M810  ; 所有異常
      OUT     T9 K10  ; 異常延時
1163  LD      SM412  ; 1sec    時鐘脈衝
      OR      M305  ; 靜音訊號
      AND     T9  ; 異常延時
      OUT     M59  ; 警報復歸LP
; //Output
1173  LD      M203  ; 恆溫訊號中
      LD      M202  ; 升溫訊號
      OR      M208  ; 降溫啟動
      AND     SM412  ; 1sec    時鐘脈衝
      ORB
      AND     M50  ; 自動模式KP
      AND     M51  ; 自動啟動KP
      AND     M200  ; <自動>  循環風車啟動
      ANI     M810  ; 所有異常
      OUT     Y0  ; 三色燈  綠燈
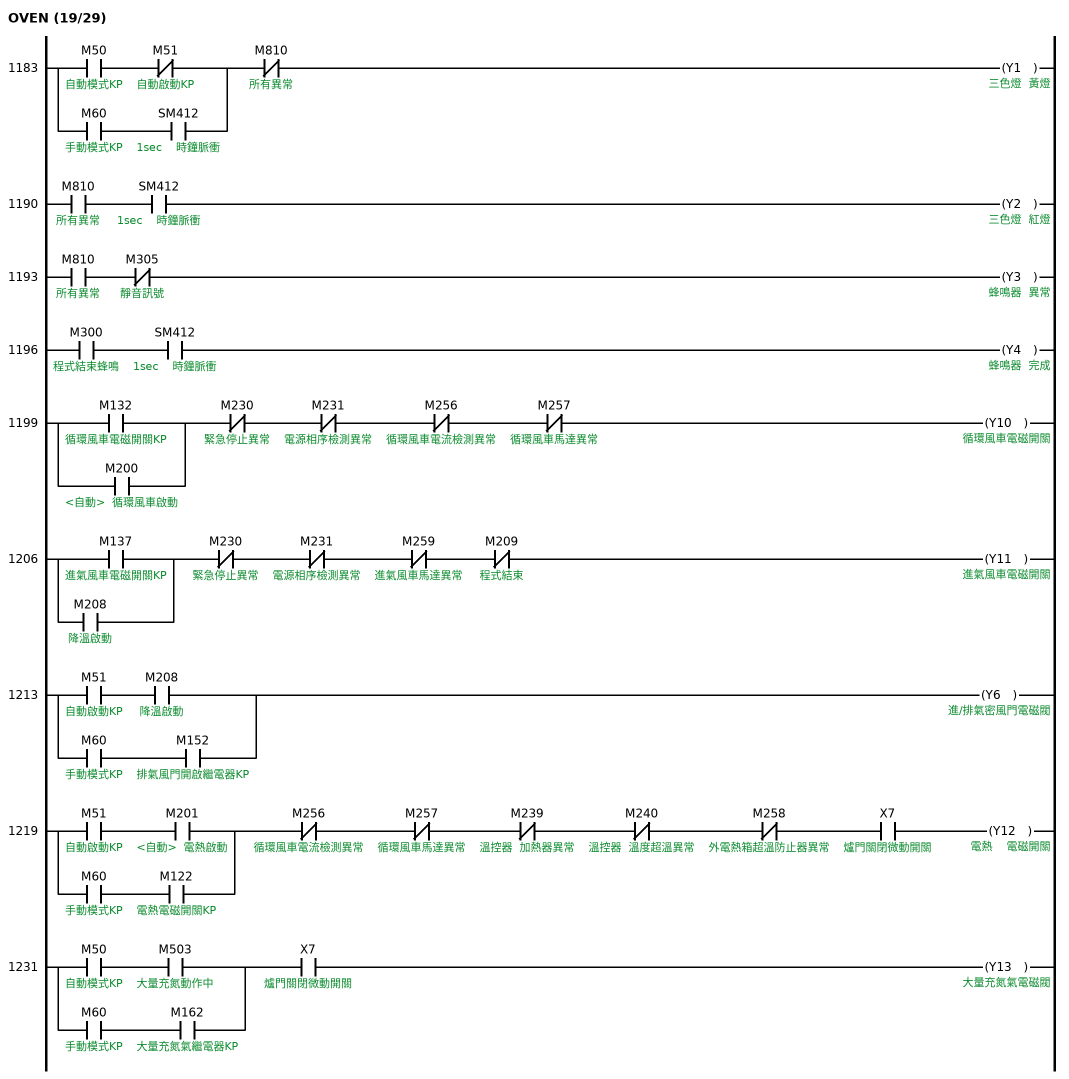
1183  LD      M50  ; 自動模式KP
      ANI     M51  ; 自動啟動KP
      LD      M60  ; 手動模式KP
      AND     SM412  ; 1sec    時鐘脈衝
      ORB
      ANI     M810  ; 所有異常
      OUT     Y1  ; 三色燈  黃燈
1190  LD      M810  ; 所有異常
      AND     SM412  ; 1sec    時鐘脈衝
      OUT     Y2  ; 三色燈  紅燈
1193  LD      M810  ; 所有異常
      ANI     M305  ; 靜音訊號
      OUT     Y3  ; 蜂鳴器  異常
1196  LD      M300  ; 程式結束蜂鳴
      AND     SM412  ; 1sec    時鐘脈衝
      OUT     Y4  ; 蜂鳴器  完成
1199  LD      M132  ; 循環風車電磁開關KP
      OR      M200  ; <自動>  循環風車啟動
      ANI     M230  ; 緊急停止異常
      ANI     M231  ; 電源相序檢測異常
      ANI     M256  ; 循環風車電流檢測異常
      ANI     M257  ; 循環風車馬達異常
      OUT     Y10  ; 循環風車電磁開關
1206  LD      M137  ; 進氣風車電磁開關KP
      OR      M208  ; 降溫啟動
      ANI     M230  ; 緊急停止異常
      ANI     M231  ; 電源相序檢測異常
      ANI     M259  ; 進氣風車馬達異常
      ANI     M209  ; 程式結束
      OUT     Y11  ; 進氣風車電磁開關
1213  LD      M51  ; 自動啟動KP
      AND     M208  ; 降溫啟動
      LD      M60  ; 手動模式KP
      AND     M152  ; 排氣風門開啟繼電器KP
      ORB
      OUT     Y6  ; 進/排氣密風門電磁閥
1219  LD      M51  ; 自動啟動KP
      AND     M201  ; <自動>  電熱啟動
      LD      M60  ; 手動模式KP
      AND     M122  ; 電熱電磁開關KP
      ORB
      ANI     M256  ; 循環風車電流檢測異常
      ANI     M257  ; 循環風車馬達異常
      ANI     M239  ; 溫控器  加熱器異常
      ANI     M240  ; 溫控器  溫度超溫異常
      ANI     M258  ; 外電熱箱超溫防止器異常
      AND     X7  ; 爐門關閉微動開關
      OUT     Y12  ; 電熱    電磁開關
1231  LD      M50  ; 自動模式KP
      AND     M503  ; 大量充氮動作中
      LD      M60  ; 手動模式KP
      AND     M162  ; 大量充氮氣繼電器KP
      ORB
      AND     X7  ; 爐門關閉微動開關
      OUT     Y13  ; 大量充氮氣電磁閥
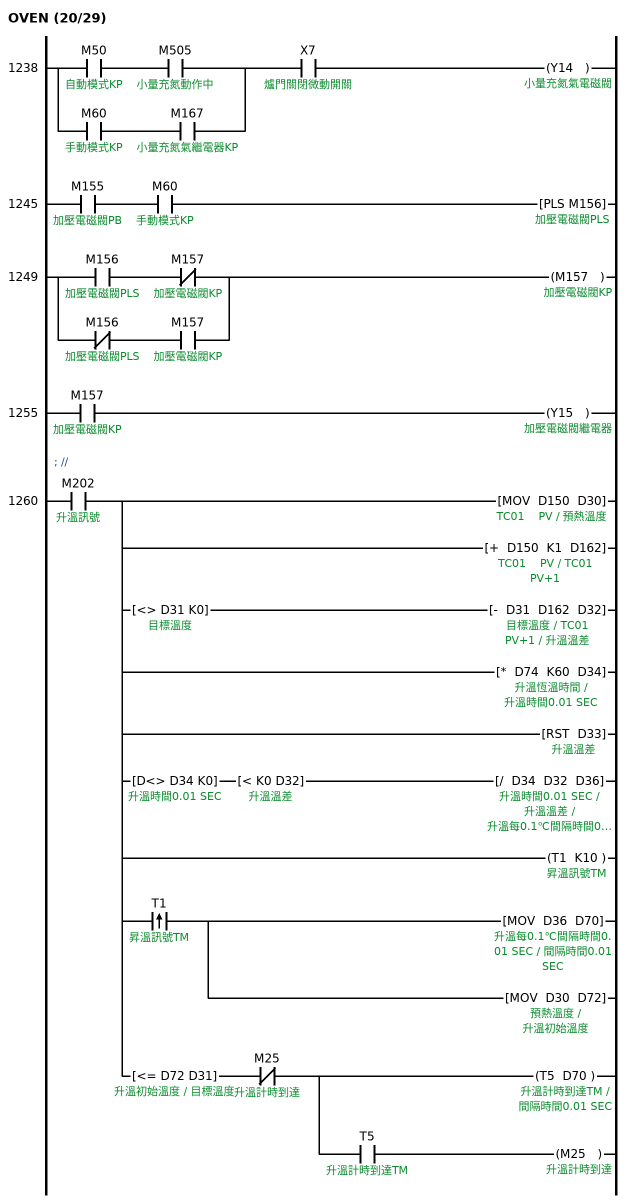
1238  LD      M50  ; 自動模式KP
      AND     M505  ; 小量充氮動作中
      LD      M60  ; 手動模式KP
      AND     M167  ; 小量充氮氣繼電器KP
      ORB
      AND     X7  ; 爐門關閉微動開關
      OUT     Y14  ; 小量充氮氣電磁閥
1245  LD      M155  ; 加壓電磁閥PB
      AND     M60  ; 手動模式KP
      PLS     M156  ; 加壓電磁閥PLS
1249  LD      M156  ; 加壓電磁閥PLS
      ANI     M157  ; 加壓電磁閥KP
      LDI     M156  ; 加壓電磁閥PLS
      AND     M157  ; 加壓電磁閥KP
      ORB
      OUT     M157  ; 加壓電磁閥KP
1255  LD      M157  ; 加壓電磁閥KP
      OUT     Y15  ; 加壓電磁閥繼電器
; //
1260  LD      M202  ; 升溫訊號
      MOV     D150 D30  ; 預熱溫度
      +       D150 K1 D162  ; TC01    PV+1
      MPS
      AND<>   D31 K0  ; 目標溫度
      -       D31 D162 D32  ; 升溫溫差
      MPP
      *       D74 K60 D34  ; 升溫時間0.01 SEC
      RST     D33  ; 升溫溫差
      MPS
      ANDD<>  D34 K0  ; 升溫時間0.01 SEC
      AND<    K0 D32  ; 升溫溫差
      /       D34 D32 D36  ; 升溫每0.1℃間隔時間0.01 SEC
      MPP
      OUT     T1 K10  ; 昇溫訊號TM
      MPS
      ANDP    T1  ; 昇溫訊號TM
      MOV     D36 D70  ; 間隔時間0.01 SEC
      MOV     D30 D72
      MPP
      AND<=   D72 D31  ; 升溫初始溫度 / 目標溫度
      ANI     M25  ; 升溫計時到達
      OUT     T5 D70  ; 升溫計時到達TM / 間隔時間0.01 SEC
      AND     T5  ; 升溫計時到達TM
      OUT     M25  ; 升溫計時到達
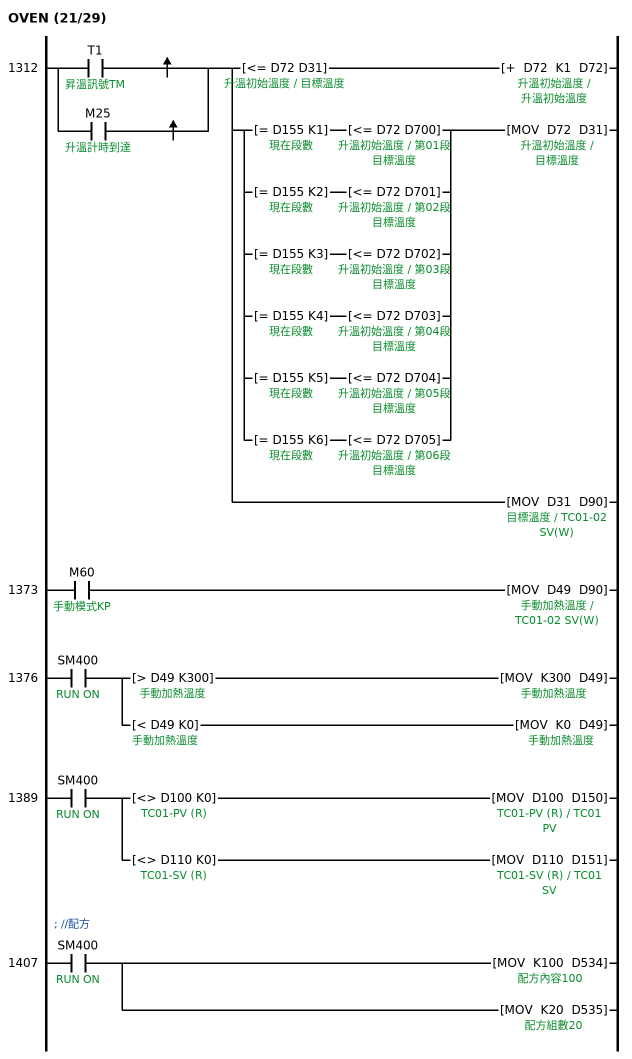
1312  LD      T1  ; 昇溫訊號TM
      MEP
      LD      M25  ; 升溫計時到達
      MEP
      ORB
      MPS
      AND<=   D72 D31  ; 升溫初始溫度 / 目標溫度
      +       D72 K1 D72
      MRD
      LD=     D155 K1  ; 現在段數
      AND<=   D72 D700  ; 升溫初始溫度 / 第01段  目標溫度
      LD=     D155 K2  ; 現在段數
      AND<=   D72 D701  ; 升溫初始溫度 / 第02段  目標溫度
      ORB
      LD=     D155 K3  ; 現在段數
      AND<=   D72 D702  ; 升溫初始溫度 / 第03段  目標溫度
      ORB
      LD=     D155 K4  ; 現在段數
      AND<=   D72 D703  ; 升溫初始溫度 / 第04段  目標溫度
      ORB
      LD=     D155 K5  ; 現在段數
      AND<=   D72 D704  ; 升溫初始溫度 / 第05段  目標溫度
      ORB
      LD=     D155 K6  ; 現在段數
      AND<=   D72 D705  ; 升溫初始溫度 / 第06段  目標溫度
      ORB
      ANB
      MOV     D72 D31
      MPP
      MOV     D31 D90  ; TC01-02 SV(W)
1373  LD      M60  ; 手動模式KP
      MOV     D49 D90  ; 手動加熱溫度
1376  LD      SM400  ; RUN ON
      MPS
      AND>    D49 K300  ; 手動加熱溫度
      MOV     K300 D49
      MPP
      AND<    D49 K0  ; 手動加熱溫度
      MOV     K0 D49
1389  LD      SM400  ; RUN ON
      MPS
      AND<>   D100 K0  ; TC01-PV (R)
      MOV     D100 D150
      MPP
      AND<>   D110 K0  ; TC01-SV (R)
      MOV     D110 D151  ; TC01    SV
; //配方
1407  LD      SM400  ; RUN ON
      MOV     K100 D534  ; 配方內容100
      MOV     K20 D535  ; 配方組數20
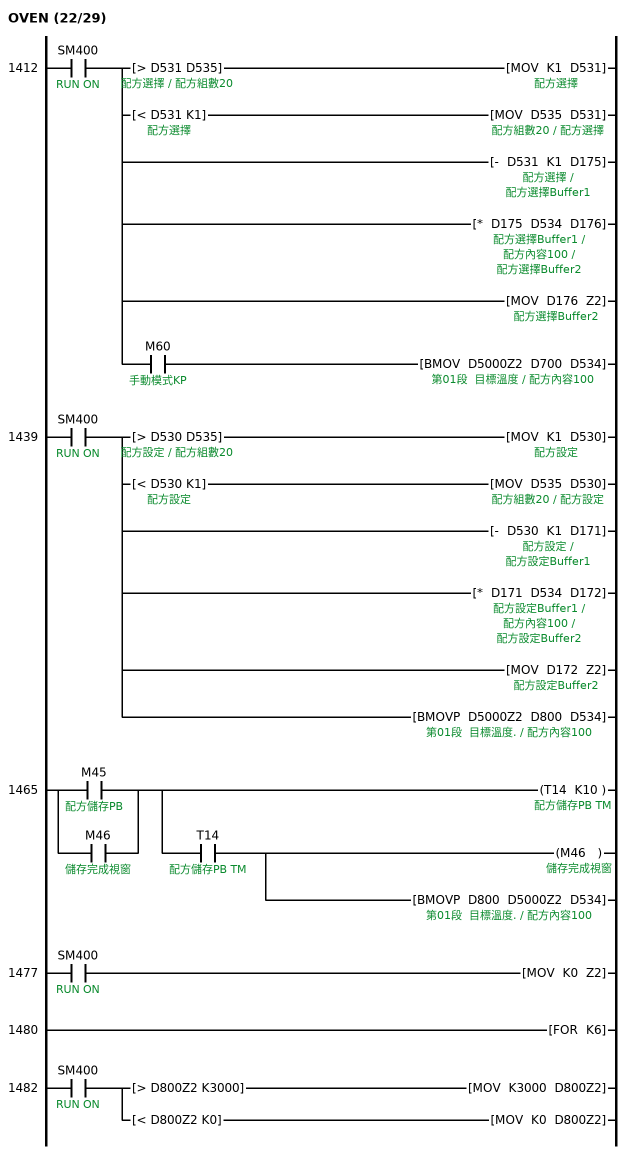
1412  LD      SM400  ; RUN ON
      MPS
      AND>    D531 D535  ; 配方選擇 / 配方組數20
      MOV     K1 D531
      MRD
      AND<    D531 K1  ; 配方選擇
      MOV     D535 D531
      MPP
      -       D531 K1 D175  ; 配方選擇Buffer1
      *       D175 D534 D176  ; 配方選擇Buffer2
      MOV     D176 Z2
      AND     M60  ; 手動模式KP
      BMOV    D5000Z2 D700 D534
1439  LD      SM400  ; RUN ON
      MPS
      AND>    D530 D535  ; 配方設定 / 配方組數20
      MOV     K1 D530
      MRD
      AND<    D530 K1  ; 配方設定
      MOV     D535 D530
      MPP
      -       D530 K1 D171  ; 配方設定Buffer1
      *       D171 D534 D172  ; 配方設定Buffer2
      MOV     D172 Z2
      BMOVP   D5000Z2 D800 D534  ; 第01段  目標溫度.
1465  LD      M45  ; 配方儲存PB
      OR      M46  ; 儲存完成視窗
      OUT     T14 K10  ; 配方儲存PB TM
      AND     T14  ; 配方儲存PB TM
      OUT     M46  ; 儲存完成視窗
      BMOVP   D800 D5000Z2 D534
1477  LD      SM400  ; RUN ON
      MOV     K0 Z2
1480  FOR     K6
1482  LD      SM400  ; RUN ON
      MPS
      AND>    D800Z2 K3000
      MOV     K3000 D800Z2
      MPP
      AND<    D800Z2 K0
      MOV     K0 D800Z2
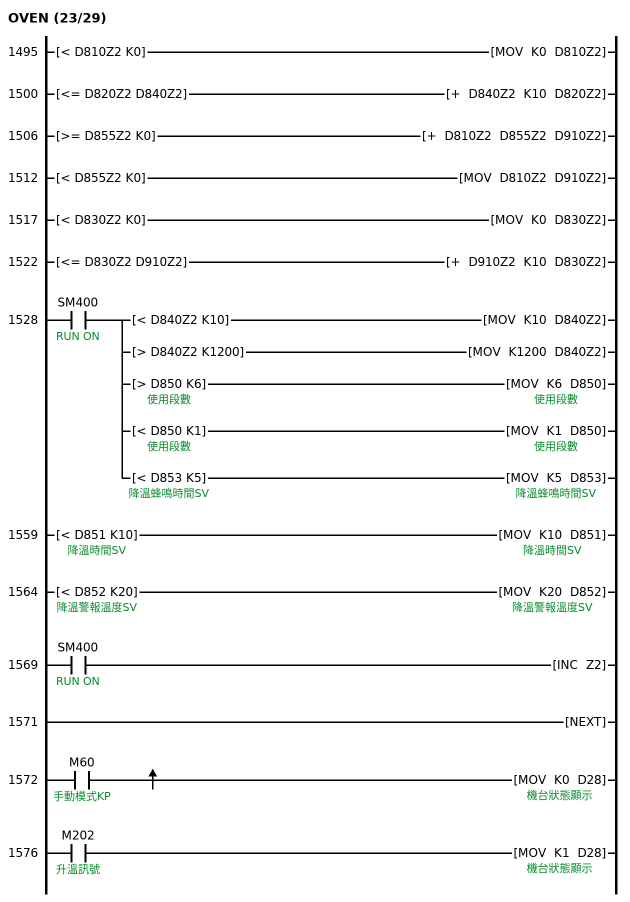
1495  LD<     D810Z2 K0
      MOV     K0 D810Z2
1500  LD<=    D820Z2 D840Z2
      +       D840Z2 K10 D820Z2
1506  LD>=    D855Z2 K0
      +       D810Z2 D855Z2 D910Z2
1512  LD<     D855Z2 K0
      MOV     D810Z2 D910Z2
1517  LD<     D830Z2 K0
      MOV     K0 D830Z2
1522  LD<=    D830Z2 D910Z2
      +       D910Z2 K10 D830Z2
1528  LD      SM400  ; RUN ON
      MPS
      AND<    D840Z2 K10
      MOV     K10 D840Z2
      MRD
      AND>    D840Z2 K1200
      MOV     K1200 D840Z2
      MRD
      AND>    D850 K6  ; 使用段數
      MOV     K6 D850
      MRD
      AND<    D850 K1  ; 使用段數
      MOV     K1 D850
      MPP
      AND<    D853 K5  ; 降溫蜂鳴時間SV
      MOV     K5 D853
1559  LD<     D851 K10  ; 降溫時間SV
      MOV     K10 D851
1564  LD<     D852 K20  ; 降溫警報溫度SV
      MOV     K20 D852
1569  LD      SM400  ; RUN ON
      INC     Z2
1571  NEXT
1572  LD      M60  ; 手動模式KP
      MEP
      MOV     K0 D28  ; 機台狀態顯示
1576  LD      M202  ; 升溫訊號
      MOV     K1 D28
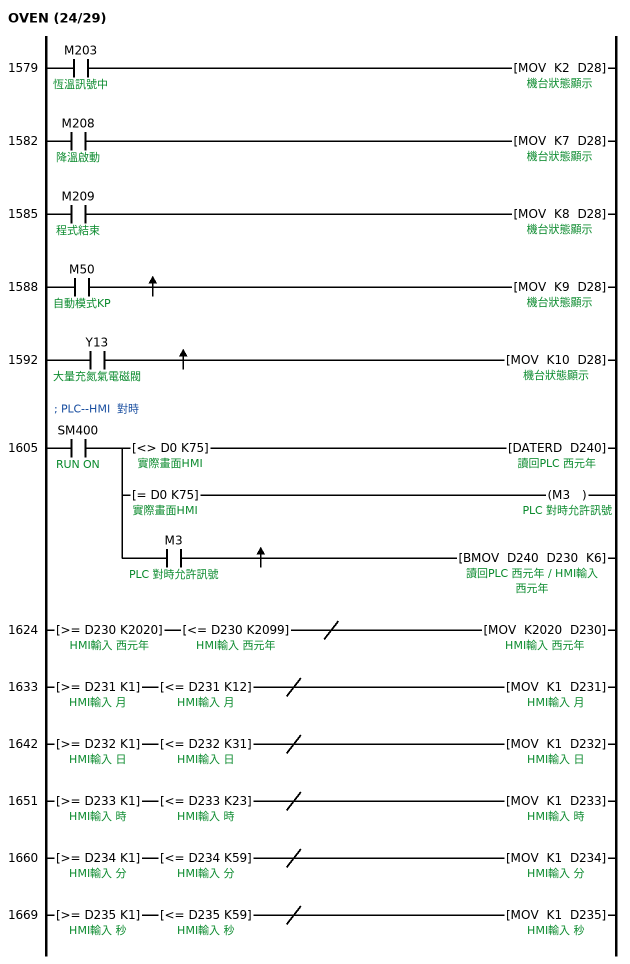
1579  LD      M203  ; 恆溫訊號中
      MOV     K2 D28
1582  LD      M208  ; 降溫啟動
      MOV     K7 D28
1585  LD      M209  ; 程式結束
      MOV     K8 D28
1588  LD      M50  ; 自動模式KP
      MEP
      MOV     K9 D28
1592  LD      Y13  ; 大量充氮氣電磁閥
      MEP
      MOV     K10 D28
; PLC--HMI  對時
1605  LD      SM400  ; RUN ON
      MPS
      AND<>   D0 K75  ; 實際畫面HMI
      DATERD  D240  ; 讀回PLC 西元年
      MRD
      AND=    D0 K75  ; 實際畫面HMI
      OUT     M3  ; PLC 對時允許訊號
      MPP
      AND     M3  ; PLC 對時允許訊號
      MEP
      BMOV    D240 D230 K6  ; HMI輸入 西元年
1624  LD>=    D230 K2020  ; HMI輸入 西元年
      AND<=   D230 K2099  ; HMI輸入 西元年
      INV
      MOV     K2020 D230
1633  LD>=    D231 K1  ; HMI輸入 月
      AND<=   D231 K12  ; HMI輸入 月
      INV
      MOV     K1 D231
1642  LD>=    D232 K1  ; HMI輸入 日
      AND<=   D232 K31  ; HMI輸入 日
      INV
      MOV     K1 D232
1651  LD>=    D233 K1  ; HMI輸入 時
      AND<=   D233 K23  ; HMI輸入 時
      INV
      MOV     K1 D233
1660  LD>=    D234 K1  ; HMI輸入 分
      AND<=   D234 K59  ; HMI輸入 分
      INV
      MOV     K1 D234
1669  LD>=    D235 K1  ; HMI輸入 秒
      AND<=   D235 K59  ; HMI輸入 秒
      INV
      MOV     K1 D235
